// TwinCAT 3 PLC project MS
// ProgramVersion: 3.1.4024.0
// libraries:
//   Tc2_ControllerToolbox, * (Beckhoff Automation GmbH)
//   Tc2_ModbusRTU, * (Beckhoff Automation GmbH)
//   Tc2_SerialCom, * (Beckhoff Automation GmbH)
//   Tc2_Standard, * (Beckhoff Automation GmbH)
//   Tc2_System, * (Beckhoff Automation GmbH)
//   Tc2_Utilities, * (Beckhoff Automation GmbH)
//   Tc3_Module, * (Beckhoff Automation GmbH)
// project tree:
//   DATA TYPES/MODUELS/ ST_GAS_CABINET.TcDUT, ST_MAIN_MODULE.TcDUT (not stored), ST_NOTIFICATION.TcDUT (not stored), ST_NOTIFICATION_MESSAGE.TcDUT, ST_REACTOR_CABINET.TcDUT (not stored), ST_SEQUENCE.TcDUT (not stored), ST_SOL_VALVE.TcDUT, ST_TEMP_CONTROLLER.TcDUT (not stored), ST_THROTTLE_VALVE.TcDUT (not stored)
//   DATA TYPES/PARTS/ ST_ANALOG_PART.TcDUT (not stored), ST_DIGITAL_PART.TcDUT (not stored), ST_SEQUENCE_PART.TcDUT (not stored)
//   DEVICE/LINE HEATER/ FB_LINE_HEATER_MANAGER.TcPOU, FB_Modbus_Send_FIFO.TcPOU, FB_TEMP_RAMPING.TcPOU (not stored)
//   DEVICE/LINE HEATER/FUNCTION/ F_Temp_Write_Set_Point.TcPOU, F_Temp_Write_Value.TcPOU (not stored)
//   DEVICE/ ST_LineHeater_Data.TcDUT (not stored), ST_Modbus_Send_Frame.TcDUT (not stored)
//   DUTs/DUTs/ENUM/ E_aAnalogInputIO_Index.TcDUT, E_AlarmList.TcDUT (not stored), E_AlarmSetValue.TcDUT, E_InputState.TcDUT (not stored), E_Interlock.TcDUT (not stored), E_Morning_Index.TcDUT (not stored), E_WarningList.TcDUT
//   DUTs/DUTs/ F_GetReal_USINT.TcDUT (not stored)
//   DUTs/ E_ControlMode.TcDUT (not stored), E_RampGeneratorState.TcDUT (not stored), E_RecipeRun.TcDUT (not stored), E_RecipeRunETMode.TcDUT (not stored), E_TowerLamp.TcDUT (not stored), OperationMode.TcDUT, outWord.TcDUT (not stored), RampGeneratorInput.TcDUT (not stored), RecipeRunET.TcDUT (not stored), RecipeStep.TcDUT, ScaleFactor.TcDUT (not stored)
//   FUNCTION/ BOOL_TO_STRING_LHeaterON.TcPOU (not stored), CheckRangeSigned.TcPOU (not stored), CheckRangeUnsigned.TcPOU (not stored), FB_TON_Pausable.TcPOU (not stored), F_GetDorPressure.TcPOU (not stored), F_State_All_Valve_Vent.TcPOU, HEXSTR_TO_REAL_LHeaterPV.TcPOU, Real_To_String_LineHeater.TcPOU (not stored), Real_To_String_ThermalBath.TcPOU (not stored), USINT_TO_WORD_Bit.TcPOU (not stored), USINT_TO_WORD_jh.TcPOU (not stored), WORD_TO_USINT_Bit.TcPOU (not stored)
//   GVLs/ GVL_COMMAND_FROM_UI.TcGVL, GVL_CONSTANT.TcGVL (not stored), GVL_DEVICE_NET_E3508.TcGVL (not stored), GVL_DEVICE_NET_IQ_PLUS.TcGVL (not stored), GVL_IO.TcGVL (not stored), GVL.TcGVL, GVL_IO_GAS_CABINET.TcGVL (not stored), GVL_IO_REACTOR_CABINET.TcGVL (not stored), GVL_IO_VALVE.TcGVL, GVL_PERSISTENT.TcGVL, GVL_SEQUENCE.TcGVL, GVL_Serial.TcGVL, RCP.TcGVL (not stored)
//   / PlcTask.TcTTO
//   POUs/ FB_AnalogDeviceRampControl.TcPOU (not stored), FB_ControlRampGenerator.TcPOU, FB_DeviationCheck.TcPOU (not stored), FB_FaultCheck.TcPOU (not stored), FB_OverLimitCheck.TcPOU (not stored), FB_RecipeAnalogControlInputSequencer.TcPOU, F_StopAnalogRamping_ForRecipe.TcPOU (not stored), FB_SensorLimitCheck.TcPOU (not stored), FB_ValveControl.TcPOU, F_ResetTimersAndRCPTimes.TcPOU (not stored), MAIN.TcPOU, P11_E3508.TcPOU (not stored), P12_IQ_PLUS.TcPOU (not stored), P13_LineHeater.TcPOU (not stored), P14_ThermalBath.TcPOU (not stored), P15_RotationOperation.TcPOU (not stored), P16_CoverOperation.TcPOU, P17_DOROperation.TcPOU (not stored), P22_Background_ThermalBath.TcPOU (not stored), P30_ManualControl.TcPOU, P31_PriorityControl.TcPOU (not stored), P50_RecipeControl.TcPOU, P60_UpdatePV.TcPOU, P70_Interface.TcPOU, P90_Interlock.TcPOU (not stored), P91_Monitoring.TcPOU, P92_Maintenance.TcPOU (not stored)
//   POUs/FUNCTION/ FB_RINGBUFFER.TcPOU (not stored), F_StateValve_Process_Source.TcPOU (not stored), F_StateValve_Process.TcPOU (not stored)
//   POUs/VARIABLE_LINK/ F_Variable_DeviceLink.TcPOU (not stored), F_Variable_Valve.TcPOU (not stored), F_Variable_FromUI.TcPOU, F_Variable_FromUI_Interlock.TcPOU (not stored), F_Variable_TODevice.TcPOU, F_Variable_ToUI_InputState.TcPOU (not stored)

CONFIGURATION MS
    RESOURCE PLC ON TwinCAT3
        TASK PlcTask(INTERVAL := T#10ms, PRIORITY := 20);
        PROGRAM MAIN WITH PlcTask : MAIN;
    END_RESOURCE
END_CONFIGURATION

// ---- DATA TYPES/MODUELS/ST_GAS_CABINET.TcDUT
TYPE ST_GAS_CABINET :
STRUCT
	DI_01_ResetButton :ST_DIGITAL_PART;
	DI_01_GasCabinetLampButton :ST_DIGITAL_PART;
	DI_01_PneumaticPressureSensor :ST_DIGITAL_PART;
	DI_01_GasCabinetDoorClose :ST_DIGITAL_PART;
	DI_01_ControlCabinetDoorClose :ST_DIGITAL_PART;
	DI_01_SMPS_1Alarm :ST_DIGITAL_PART;
	DI_01_SMPS_2Alarm :ST_DIGITAL_PART;
	DI_01_SMPS_3Alarm :ST_DIGITAL_PART;
	
	DI_02_SMPS_4Alarm :ST_DIGITAL_PART;
	DI_02_GraphiteHeaterELCB :ST_DIGITAL_PART;
	DI_02_ThermalBathsELCB :ST_DIGITAL_PART;
	DI_02_VacuumPumpELCB :ST_DIGITAL_PART;
	DI_02_LineHeatersELCB :ST_DIGITAL_PART;
	DI_02_RotationMotorCP :ST_DIGITAL_PART;
	DI_02_CoverLiftMotorCP :ST_DIGITAL_PART;
	DI_02_T_VCP :ST_DIGITAL_PART;
	
	DI_03_GasDetectorCP :ST_DIGITAL_PART;
	DI_03_CabinetLampsCP :ST_DIGITAL_PART;
	DI_03_MFCPowerCP :ST_DIGITAL_PART;
	DI_03_LineHeater_1CP :ST_DIGITAL_PART;
	DI_03_LineHeater_2CP :ST_DIGITAL_PART;
	DI_03_LineHeater_3CP :ST_DIGITAL_PART;
	
	DI_03_LineHeater_4CP :ST_DIGITAL_PART;
	DI_03_LineHeater_5CP :ST_DIGITAL_PART;
	DI_04_LineHeater_6CP :ST_DIGITAL_PART;
	DI_04_LineHeater_7CP :ST_DIGITAL_PART;
	DI_04_LineHeater_8CP :ST_DIGITAL_PART;
	DI_04_GasDetectorH2 :ST_DIGITAL_PART;
	DI_04_GasDetectorH2S :ST_DIGITAL_PART;
	DI_04_GasDetectorH2Se :ST_DIGITAL_PART;
	DI_04_FireSensor :ST_DIGITAL_PART;
	DI_04_ExternalScrubberFault :ST_DIGITAL_PART;
	
	DI_05_ExternalH2GasCabinetFault :ST_DIGITAL_PART;
	DI_05_ExternalH2SGasCabinetFault :ST_DIGITAL_PART;
	DI_05_ExternalH2SeGasCabinetFault :ST_DIGITAL_PART;
	DI_05_ExternalUserInputAlarm :ST_DIGITAL_PART;
	DI_05_ThermalBath_1DeviationAlarm :ST_DIGITAL_PART;
	DI_05_ThermalBath_1CutOffAlarm :ST_DIGITAL_PART;
	DI_05_ThermalBath_2DeviationAlarm :ST_DIGITAL_PART;
	DI_05_ThermalBath_2CutOffAlarm :ST_DIGITAL_PART;
	
	DI_06_ThermalBath_3DeviationAlarm :ST_DIGITAL_PART;
	DI_06_ThermalBath_3CutOffAlarm :ST_DIGITAL_PART;
	DI_06_ThermalBath_4DeviationAlarm :ST_DIGITAL_PART;
	DI_06_ThermalBath_4CutOffAlarm :ST_DIGITAL_PART;
	DI_06_Spare_01 :ST_DIGITAL_PART;
	DI_06_Spare_02 :ST_DIGITAL_PART;
	DI_06_Spare_03 :ST_DIGITAL_PART;
	DI_06_Spare_04 :ST_DIGITAL_PART;
	
	DO_07_SystemPowerOffLock :ST_DIGITAL_PART;
	DO_07_GasCabinetLamp :ST_DIGITAL_PART;
	DO_07_ControlCabinetLamp :ST_DIGITAL_PART;
	DO_07_GraphiteHeaterMC :ST_DIGITAL_PART;
	DO_07_ThermalBathsMC :ST_DIGITAL_PART;
	DO_07_VacuumPumpMC :ST_DIGITAL_PART;
	DO_07_LineHeatersMC :ST_DIGITAL_PART;
	DO_07_ResetButtonLamp :ST_DIGITAL_PART;
	
	DO_08_Spare_01 :ST_DIGITAL_PART;
	DO_08_Spare_02 :ST_DIGITAL_PART;
	DO_08_Spare_03 :ST_DIGITAL_PART;
	DO_08_Spare_04 :ST_DIGITAL_PART;
	DO_08_Spare_05 :ST_DIGITAL_PART;
	DO_08_Spare_06 :ST_DIGITAL_PART;
	DO_08_Spare_07 :ST_DIGITAL_PART;
	DO_08_Spare_08 :ST_DIGITAL_PART;
	
	AI_09_M01_ChalcogenRunPV :ST_ANALOG_PART;
	AI_09_M02_MORunPV :ST_ANALOG_PART;
	AI_09_M03_H2SeSupplyPV :ST_ANALOG_PART;
	AI_09_M04_H2SSupplyPV :ST_ANALOG_PART;
	
	AO_10_M01_ChalcogenRunSV :ST_ANALOG_PART;
	AO_10_M02_MORunSV :ST_ANALOG_PART;
	AO_10_M03_H2SeSupplySV :ST_ANALOG_PART;
	AO_10_M04_H2SSupplySV :ST_ANALOG_PART;
	
	AI_11_M05_Source_1TMInSupplyPV :ST_ANALOG_PART;
	AI_11_M06_Source_2TMGaSupplyPV :ST_ANALOG_PART;
	AI_11_M07_Source_3DMSeSupplyPV :ST_ANALOG_PART;
	AI_11_M08_Source_4ChalcoSupplyPV :ST_ANALOG_PART;
	
	AO_12_M05_Source_1TMInSupplySV :ST_ANALOG_PART;
	AO_12_M06_Source_2TMGaSupplySV :ST_ANALOG_PART;
	AO_12_M07_Source_3DMSeSupplySV :ST_ANALOG_PART;
	AO_12_M08_Source_4ChalcoSupplySV :ST_ANALOG_PART;
	
	AI_13_M09_LinerPurgePV :ST_ANALOG_PART;
	AI_13_M10_HeaterPurgePV :ST_ANALOG_PART;
	AI_13_M11_ChalcogenVentPV :ST_ANALOG_PART;
	AI_13_M12_MOVentPV :ST_ANALOG_PART;
	
	AO_14_M09_LinerPurgeSV :ST_ANALOG_PART;
	AO_14_M10_HeaterPurgeSV :ST_ANALOG_PART;
	AO_14_M11_ChalcogenVentSV :ST_ANALOG_PART;
	AO_14_M12_MOVentSV :ST_ANALOG_PART;
	
	AI_15_E01Source_1TMInPressurePV :ST_ANALOG_PART;
	AI_15_E02Source_2TMGaPressurePV :ST_ANALOG_PART;
	AI_15_E03Source_3DMSePressurePV :ST_ANALOG_PART;
	AI_15_E04Source_4ChalcoPressurePV :ST_ANALOG_PART;
	
	AO_16_E01Source_1TMInPressureSV :ST_ANALOG_PART;
	AO_16_E02Source_2TMGaPressureSV :ST_ANALOG_PART;
	AO_16_E03Source_3DMSePressureSV :ST_ANALOG_PART;
	AO_16_E04Source_4ChalcoPressureSV :ST_ANALOG_PART;
	
	DI_17_DP1ChalcogenDP :ST_ANALOG_PART;
	DI_17_DP2MODP :ST_ANALOG_PART;
	
	DI_18_S01N2SupplyPressPV :ST_ANALOG_PART;
	DI_18_S02H2SupplyPressPV :ST_ANALOG_PART;
	DI_18_S03H2SSupplyPressPV :ST_ANALOG_PART;
	DI_18_S04H2SeSupplyPressPV :ST_ANALOG_PART;
	
	DI_19_LineHeaterController :ST_DIGITAL_PART;
	DI_20_ThermalBathx4EA :ST_DIGITAL_PART;

END_STRUCT
END_TYPE

// ---- DATA TYPES/MODUELS/ST_NOTIFICATION_MESSAGE.TcDUT
TYPE ST_NOTIFICATION_MESSAGE :
STRUCT
	INDEX:DINT;
	TITLE:STRING(255);
	MESSAGE :STRING(255);
	NOTIFICATION_TYPE:DINT; (* NOTIFI_INTERLOCK = 1, NOTIFI_ALARM = 2, NOTIFI_MESSAGE = 3 *)
	MODULE_ID:DINT;
END_STRUCT
END_TYPE

// ---- DATA TYPES/MODUELS/ST_SOL_VALVE.TcDUT
TYPE ST_SOL_VALVE :
STRUCT
	DO_00_V01ChalcogenCarrierChange :ST_DIGITAL_PART;
	DO_00_V02MOCarreirChange :ST_DIGITAL_PART;
	DO_00_V03H2SeSourceChange :ST_DIGITAL_PART;
	DO_00_V04H2SSourceChange :ST_DIGITAL_PART;
	DO_00_V05Source_1TMInCarrierChange :ST_DIGITAL_PART;
	DO_00_V06Source_1TMInBypass :ST_DIGITAL_PART;
	DO_00_V07Source_2TMGaCarrierChange :ST_DIGITAL_PART;
	DO_00_V08Source_2TMGaBypass :ST_DIGITAL_PART;
	
	DO_00_V09Source_3DMSeCarrierChange :ST_DIGITAL_PART;
	DO_00_V10Source_3DMSeBypass :ST_DIGITAL_PART;
	DO_00_V11Source_4ChalcogenCarrierChange :ST_DIGITAL_PART;
	DO_00_V12Source_4ChalcogenBypass :ST_DIGITAL_PART;
	DO_00_V13ReactorPurgeCarrierChange :ST_DIGITAL_PART;
	DO_00_V14Source_1TMInManifoldRun :ST_DIGITAL_PART;
	DO_00_V15Source_2TMGaManifoldRun :ST_DIGITAL_PART;
	DO_00_V16Source_3DMSeManifoldRun :ST_DIGITAL_PART;
	
	DO_00_V17GasH2SeManifoldRun :ST_DIGITAL_PART;
	DO_00_V18GasH2SManifoldRun :ST_DIGITAL_PART;
	DO_00_V19Source_4ChalcogenManifoldRun :ST_DIGITAL_PART;
	DO_00_V20VentPress_Change :ST_DIGITAL_PART;
	DO_00_V21PumpByPass :ST_DIGITAL_PART;
	DO_00_V22DORVaccumON :ST_DIGITAL_PART;
	DO_00_V23DORFilling :ST_DIGITAL_PART;
	DO_00_V24Source_1LeakTest_IN :ST_DIGITAL_PART;
	
	DO_00_V25Source_1LeakTest_OUT :ST_DIGITAL_PART;
	DO_00_V26Source_2LeakTest_IN :ST_DIGITAL_PART;
	DO_00_V27Source_2LeakTest_OUT :ST_DIGITAL_PART;
	DO_00_V28Source_3LeakTest_IN :ST_DIGITAL_PART;
	DO_00_V29Source_3LeakTest_OUT :ST_DIGITAL_PART;
	DO_00_V30Source_4LeakTest_IN :ST_DIGITAL_PART;
	DO_00_V31Source_4LeakTest_OUT :ST_DIGITAL_PART;
	DO_00_V32SourceVacuumON :ST_DIGITAL_PART;
	
END_STRUCT
END_TYPE

// ---- DUTs/DUTs/ENUM/E_aAnalogInputIO_Index.TcDUT
{attribute 'qualified_only'}
{attribute 'strict'}
{attribute 'to_string'}
TYPE E_aAnalogInputIO_Index :
(
	E_PV_MFC_01 :=1,
	E_PV_MFC_02 :=2,
	E_PV_MFC_03 :=3,
	E_PV_MFC_04 :=4,
	E_PV_MFC_05 :=5,
	E_PV_MFC_06 :=6,
	E_PV_MFC_07 :=7,
	E_PV_MFC_08 :=8,
	E_PV_MFC_09 :=9,
	E_PV_MFC_10 :=10,
	E_PV_MFC_11 :=11,
	E_PV_MFC_12 :=12,
	E_PV_EPC_01 :=13,
	E_PV_EPC_02 :=14,
	E_PV_EPC_03 :=15,
	E_PV_EPC_04 :=16,
	E_PV_Susceptor_Temp:=17,
	E_PV_Reactor_Pressure:=18,
	E_PV_susceptorRotation:=19,
	E_PV_Ultimate_Pressure:=20,
	E_PV_Exhaust_Pressure:=21,
	E_PV_DOR_PRESSURE:=22,
	E_PV_GAS_Pressure_N2:=23,
	E_PV_GAS_Pressure_H2:=24,
	E_PV_GAS_Pressure_H2S:=25,
	E_PV_GAS_Pressure_H2Se:=26,
	E_PV_CoolingWafer_SH:=27
);
END_TYPE

// ---- DUTs/DUTs/ENUM/E_AlarmSetValue.TcDUT
{attribute 'qualified_only'}
{attribute 'strict'}
{attribute 'to_string'}
TYPE E_AlarmSetValue :
(
//	E_AS_Alarm_Deviation:=1,
//	E_AS_Warning_Deviation,
//	E_AS_DelayTime_Analog,
//	E_AS_DelayTime_Digital,
//	E_AS_Process_Gas_Pressure_Alarm,
//	E_AS_Process_Gas_Pressure_Warning,
//	E_AS_CWTemp_SH_ALARM,
//	E_AS_CWTemp_SH_WARNING,
//	E_AS_CWTemp_COIL_ALARM,
//	E_AS_CWTemp_COIL_WARNING,
//	E_AS_SUSCEPTOR_OVER_TEMP,
//	E_AS_REACTOR_OVRE_PRESSURE,
//	E_AS_CAN_OPEN_TEMP,
//	E_AS_CAN_OPEN_REACTOR_PRESSURE,
//	E_AS_DOR_Pressure_Limit,
//	E_AS_DOR_RerayCount,
	E_AS_END
);
END_TYPE

// ---- DUTs/DUTs/ENUM/E_WarningList.TcDUT
{attribute 'qualified_only'}
{attribute 'strict'}
{attribute 'to_string'}
TYPE E_WarningList :
(
	E_WarningList_GasPressure_Low_N2:=1,
	E_WarningList_GasPressureLowN2,
	E_WarningList_GasPressureLowH2,
	E_WarningList_GasPressureLowNH3,
	E_WarningList_GasPressureLowSiH4,
	E_WarningList_CWTemperatureHighSH,
	E_WarningList_CWTemperatureHighCoil,
	E_WarningList_SusceptorOverTemperature,
	E_WarningList_ReactorOverPressure,
	E_WarningList_PneumaticPressureLow,
	E_WarningList_CoolingWaterLow,
	E_WarningList_InductionHeaterFault,
	E_WarningList_RotationMotorFault,
	E_WarningList_VacuumPumpFault,
	E_WarningList_GasCabinetDoorOpen,
	E_WarningList_ReactorCabinetDoorOpen,
	E_WarningList_SusceptorTemperatureDeviation,
	E_WarningList_ReactorPressureDeviation,
	E_WarningList_SusceptorRotationDeviation,
	E_WarningList_MORunDeviation,
	E_WarningList_HydRunDeviation,
	E_WarningList_NH3LargeINDeviation,
	E_WarningList_NH3SmallINDeviation,
	E_WarningList_SiHINDeviation,
	E_WarningList_SiHDilutionDeviation,
	E_WarningList_SiHDilutedDeviation,
	E_WarningList_TEBBubblingDeviation,
	E_WarningList_TMAlBubblingDeviation,
	E_WarningList_TMInBubblingDeviation,
	E_WarningList_TMGaBubblingDeviation,
	E_WarningList_DTMGaBubblingDeviation,
	E_WarningList_DTMGaDilutionDeviation,
	E_WarningList_DTMGaDilutedDeviation,
	E_WarningList_Cp2MgBubblingDeviation,
	E_WarningList_ReactorPurgeDeviation,
	E_WarningList_RotationSealPurgeDeviation,
	E_WarningList_MOVentDeviation,
	E_WarningList_HydVentDeviation,
	E_WarningList_SiH4PressureDeviation,
	E_WarningList_TEBPressureDeviation,
	E_WarningList_TMAlPressureDeviation,
	E_WarningList_TMInPressureDeviation,
	E_WarningList_TMGaPressureDeviation,
	E_WarningList_DTMGaPressureDeviation,
	E_WarningList_Cp2MgPressureDeviation,
	E_WarningList_END

);
END_TYPE

// ---- DUTs/OperationMode.TcDUT
{attribute 'qualified_only'}
{attribute 'strict'}
{attribute 'to_string'}
TYPE OperationMode :
(
	Manual := 0,
	Recipe := 1,
	Priority := 2
);
END_TYPE

// ---- DUTs/RecipeStep.TcDUT
TYPE RecipeStep :
STRUCT
	sRecipe : STRING(81);
	iRecipe : ARRAY[1..5] OF INT; //Reactor Condition
	rRecipe : ARRAY[1..GVL_CONSTANT.NumAnalogController] OF REAL; //MFC, EPC Data
	cTemp 	: REAL := 0; 	
	dRecipe : DWORD; //Valve Data
END_STRUCT
END_TYPE

// ---- GVLs/GVL_COMMAND_FROM_UI.TcGVL
{attribute 'qualified_only'}
VAR_GLOBAL
	
	//GVL_IO.aOutputCmd[1].
	
	CMD_HEATER_MAIN_MC_ON:BOOL;  //[1].0
	CMD_THERMAL_BACH_MC_ON:BOOL;//[1].1
	CMD_VACUUM_PUMP_MC_ON:BOOL;//[1].2
	CMD_LINE_HEATER_MC_ON:BOOL;//[1].3
	CMD_SPARE_1_4:BOOL;//[1].4
	CMD_SPARE_1_5:BOOL;//[1].5
	CMD_VACUUM_PUMP_ON:BOOL;//[1].6
	CMD_VACUUM_PUMP_RESET:BOOL;//[1].7
	CMD_ROTATION_START:BOOL;//[1].8
	CMD_ROTATION_RESET:BOOL;//[1].9
	CMD_MAIN_POWER_RESET:BOOL;//[1].10
	
	CMD_E3508_MAN_AUTO:BOOL;//[1].11
	CMD_THROTTLE_PRESSURE_POSITION_MODE:BOOL;//[1].12
	CMD_THROTTLE_OUTPUT_MODE:USINT;//[2]	
END_VAR

// ---- GVLs/GVL.TcGVL
{attribute 'qualified_only'}
VAR_GLOBAL
	MainModule:ST_MAIN_MODULE;
	fbLineHeater_Manager:FB_LINE_HEATER_MANAGER;
	
	RotationResetTon: TON;
END_VAR

// ---- GVLs/GVL_IO_VALVE.TcGVL
{attribute 'qualified_only'}
VAR_GLOBAL
	DO_00_V01ChalcogenCarrierChange AT%Q*:BOOL;
	DO_00_V02MOCarreirChange AT%Q*:BOOL;
	DO_00_V03H2SeSourceChange AT%Q*:BOOL;
	DO_00_V04H2SSourceChange AT%Q*:BOOL;
	DO_00_V05Source_1TMInCarrierChange AT%Q*:BOOL;
	DO_00_V06Source_1TMInBypass AT%Q*:BOOL;
	DO_00_V07Source_2TMGaCarrierChange AT%Q*:BOOL;
	DO_00_V08Source_2TMGaBypass AT%Q*:BOOL;
	DO_00_V09Source_3DMSeCarrierChange AT%Q*:BOOL;
	DO_00_V10Source_3DMSeBypass AT%Q*:BOOL;
	DO_00_V11Source_4ChalcogenCarrierChange AT%Q*:BOOL;
	DO_00_V12Source_4ChalcogenBypass AT%Q*:BOOL;
	DO_00_V13ReactorPurgeCarrierChange AT%Q*:BOOL;
	DO_00_V14Source_1TMInManifoldRun AT%Q*:BOOL;
	DO_00_V15Source_2TMGaManifoldRun AT%Q*:BOOL;
	DO_00_V16Source_3DMSeManifoldRun AT%Q*:BOOL;
	DO_00_V17GasH2SeManifoldRun AT%Q*:BOOL;
	DO_00_V18GasH2SManifoldRun AT%Q*:BOOL;
	DO_00_V19Source_4ChalcogenManifoldRun AT%Q*:BOOL;
	DO_00_V20VentPress_Change AT%Q*:BOOL;
	DO_00_V21PumpByPass AT%Q*:BOOL;
	DO_00_V22DORVaccumON AT%Q*:BOOL;
	DO_00_V23DORFilling AT%Q*:BOOL;
	DO_00_V24Source_1LeakTest_IN AT%Q*:BOOL;
	DO_00_V25Source_1LeakTest_OUT AT%Q*:BOOL;
	DO_00_V26Source_2LeakTest_IN AT%Q*:BOOL;
	DO_00_V27Source_2LeakTest_OUT AT%Q*:BOOL;
	DO_00_V28Source_3LeakTest_IN AT%Q*:BOOL;
	DO_00_V29Source_3LeakTest_OUT AT%Q*:BOOL;
	DO_00_V30Source_4LeakTest_IN AT%Q*:BOOL;
	DO_00_V31Source_4LeakTest_OUT AT%Q*:BOOL;
	DO_00_V32SourceVacuumON AT%Q*:BOOL;
END_VAR

// ---- GVLs/GVL_PERSISTENT.TcGVL
{attribute 'qualified_only'}
VAR_GLOBAL PERSISTENT
	parameter_Test:INT;
	parameter_Test_1:INT;
	parameter_Test_2:INT;
END_VAR

// ---- GVLs/GVL_SEQUENCE.TcGVL
{attribute 'qualified_only'}
VAR_GLOBAL
//	fbUpdateModue:FB_UPDATE_MODULE;
	
	fbDeviationCheck		:ARRAY[1..29] OF FB_DeviationCheck;
	fbDeviationCheck_Reactor		:ARRAY[1..3] OF FB_DeviationCheck;
	fbSensorLimitCheck		:ARRAY[1..4] OF FB_SensorLimitCheck;  // Pressure N2 H2 H2S,H2SE 
	fbSensorOverLimitCheck	:ARRAY[1..2] OF FB_OverLimitCheck;  // Over Temp  , Over Pressure  
	fbFaultCheck			:ARRAY[1..8] OF FB_FaultCheck; // CDA/CoolingWafer/Rotation Fault/Vacuum Pump Fault/Gas Cabinet Open / Reactor Door Open / Dor Fault
	fbFaultCheck_Utility	:ARRAY[1..4] OF FB_FaultCheck; //SMPS,Circuit Power , Gas Detector , External Alarm
	fbFaultCheck_Utility_CP :ARRAY[1..4] OF FB_FaultCheck; //CP
	
	FB_DOR_PRESSURE_AVG: FB_RINGBUFFER;
	FB_EXHAUST_AVG: FB_RINGBUFFER;
END_VAR

// ---- GVLs/GVL_Serial.TcGVL
{attribute 'qualified_only'}
VAR_GLOBAL
	TxBufferTB : ComBuffer; (* Receive data buffer; used with all receive function blocks *)
	RxBufferTB : ComBuffer; (* Transmit data buffer; used with all receive function blocks *)
	
	stIn_KL6031_TB AT %I*	: KL6inData22B;	(* linked to the KL6001 in the TwinCAT System Manager *)
	stOut_KL6031_TB AT %Q*	: KL6outData22B;	(* linked to the KL6001 in the TwinCAT System Manager *)	
	
	LineHeater_data_1	:ST_LineHeater_Data;
	LineHeater_data_2	:ST_LineHeater_Data;
END_VAR

// ---- POUs/MAIN.TcPOU
PROGRAM MAIN
VAR_INPUT
	controlModeCmd : E_ControlMode := E_ControlMode.Manual;
END_VAR
VAR
	controlMode	: E_ControlMode := controlModeCmd;
	prevControlMode : E_ControlMode := controlMode;
END_VAR

F_Variable_Valve();
F_Variable_DeviceLink();
F_Variable_FromUI();
F_Variable_FromUI_Interlock();
F_Variable_TODevice();
F_Variable_ToUI_InputState();
GVL.fbLineHeater_Manager(RData_Module_1=>GVL_Serial.LineHeater_data_1,RData_Module_2=>GVL_Serial.LineHeater_data_2);


P11_E3508(); //Temp Controller
P12_IQ_PLUS(); //Throttle Valve Controller
P13_LineHeater();
P14_ThermalBath();
P15_RotationOperation();
P16_CoverOperation();
P17_DOROperation();
P22_Background_ThermalBath();


IF controlMode <> E_ControlMode.Priority THEN
	IF controlMode <> controlModeCmd THEN
		IF controlModeCmd = E_ControlMode.Priority THEN
			prevControlMode := controlMode;
		END_IF
		controlMode := controlModeCmd;
	END_IF
END_IF

CASE controlMode OF
	E_ControlMode.Manual:
		P30_ManualControl();
	
	E_ControlMode.Recipe:
		P50_RecipeControl(); //레시피 콘트론
		
	E_ControlMode.Priority:
		P31_PriorityControl();
		IF P31_PriorityControl.complete = TRUE THEN
			controlMode := prevControlMode;
			controlModeCmd := controlMode;
		END_IF
END_CASE

P60_UpdatePV();
P70_Interface();
P90_Interlock();
P91_Monitoring();
P92_Maintenance();

END_PROGRAM

// ---- POUs/VARIABLE_LINK/F_Variable_FromUI.TcPOU
FUNCTION F_Variable_FromUI: BOOL


VAR
	rRotationAlarm_Reset: R_TRIG;
	
	Rotation_Shift: WORD;
END_VAR

////UI에서 Write하는 Command
//아래 MC는 Maint 모드에서만 조작 가능
//GVL_COMMAND_FROM_UI.CMD_HEATER_MAIN_MC_ON:= GVL_IO.aOutputCmd[1].0;
//GVL_COMMAND_FROM_UI.CMD_THERMAL_BACH_MC_ON:= GVL_IO.aOutputCmd[1].1;
//GVL_COMMAND_FROM_UI.CMD_VACUUM_PUMP_MC_ON:= GVL_IO.aOutputCmd[1].2;
//GVL_COMMAND_FROM_UI.CMD_LINE_HEATER_MC_ON := GVL_IO.aOutputCmd[1].3;

GVL_COMMAND_FROM_UI.CMD_VACUUM_PUMP_ON := GVL_IO.aOutputCmd[1].6;
GVL_COMMAND_FROM_UI.CMD_VACUUM_PUMP_RESET:= GVL_IO.aOutputCmd[1].7;

GVL_COMMAND_FROM_UI.CMD_ROTATION_START:= GVL_IO.aOutputCmd[1].8;
GVL_COMMAND_FROM_UI.CMD_ROTATION_RESET := GVL_IO.aOutputCmd[1].10;

//jhkang 하드웨어로 구성 되어 있어야 하는데 아직 구성 안됨 := GVL_IO.aOutputCmd[1].10;
GVL_COMMAND_FROM_UI.CMD_E3508_MAN_AUTO := GVL_IO.aOutputCmd[1].12;(*True:Manual  False:auto*)
GVL_COMMAND_FROM_UI.CMD_THROTTLE_PRESSURE_POSITION_MODE := GVL_IO.aOutputCmd[1].13;//true: Pressure False:Position

GVL_COMMAND_FROM_UI.CMD_THROTTLE_OUTPUT_MODE:= WORD_TO_USINT(GVL_IO.aOutputCmd[2]); //Throttle Valve Mode Setting 0:Normal 1:Close 2:Open 3:Hold 4:Reset

GVL_IO_GAS_CABINET.DO_07_GraphiteHeaterMC :=  GVL_COMMAND_FROM_UI.CMD_HEATER_MAIN_MC_ON;
GVL_IO_GAS_CABINET.DO_07_ThermalBathsMC :=  GVL_COMMAND_FROM_UI.CMD_THERMAL_BACH_MC_ON;
GVL_IO_GAS_CABINET.DO_07_VacuumPumpMC :=  GVL_COMMAND_FROM_UI.CMD_VACUUM_PUMP_MC_ON;
GVL_IO_GAS_CABINET.DO_07_LineHeatersMC:=  GVL_COMMAND_FROM_UI.CMD_LINE_HEATER_MC_ON;

//GVL_IO_REACTOR_CABINET.DO_05_SusceptorRotationFWD:=GVL_COMMAND_FROM_UI.CMD_ROTATION_START;

rRotationAlarm_Reset(CLK:=GVL_COMMAND_FROM_UI.CMD_ROTATION_RESET);
IF rRotationAlarm_Reset.Q THEN
	GVL_IO_REACTOR_CABINET.DO_05_SusceptorRotationAL_RST:=TRUE;
END_IF

GVL.RotationResetTon(IN:=GVL_IO_REACTOR_CABINET.DO_05_SusceptorRotationAL_RST,PT:=T#3S);

IF GVL_IO_REACTOR_CABINET.DI_02_SusceptorRotationMotorFault = TRUE OR GVL.RotationResetTon.Q THEN
	GVL.RotationResetTon(in:=FALSE);
	IF GVL_IO_REACTOR_CABINET.DO_05_SusceptorRotationAL_RST = TRUE THEN
		GVL_IO_REACTOR_CABINET.DO_05_SusceptorRotationAL_RST:=FALSE;
	END_IF
	
	IF GVL_IO.aOutputCmd[1].10 = TRUE THEN
		GVL_IO.aOutputCmd[1].10:=FALSE;
	END_IF
END_IF


	//GVL_IO_REACTOR_CABINET.DO_05_SusceptorRotationAL_RST:=GVL_COMMAND_FROM_UI.CMD_ROTATION_RESET;	
GVL_IO_REACTOR_CABINET.DO_05_VacuumPumpStart_Stop := GVL_COMMAND_FROM_UI.CMD_VACUUM_PUMP_ON;
GVL_IO_REACTOR_CABINET.DO_05_VacuumPumpReset:=GVL_COMMAND_FROM_UI.CMD_VACUUM_PUMP_RESET;

END_FUNCTION

// ---- POUs/VARIABLE_LINK/F_Variable_TODevice.TcPOU
FUNCTION F_Variable_TODevice: BOOL

;

END_FUNCTION

// ---- POUs/P16_CoverOperation.TcPOU
PROGRAM P16_CoverOperation
VAR
// 	isCoverClosed 	: BOOL;

	bCoverCP	: BOOL;
	bLowerLimit	: BOOL;
	bUpperLimit	: BOOL;
	TimerUpLED 		: TON;
	TimerUpLED_X 	: TON;
	TimerDownLED 	: TON;
	TimerDownLED_X 	: TON;
	TimerDownDelayOff 	: TON;
	(* Input *)
	bUpSwitch	: BOOL;
	bDownSwitch 	: BOOL;
	bClamp_Lock_switch: BOOL;
	bClamp_Release_switch: BOOL;
	(* Output *)
	bUpLED 		: BOOL;
	bDownLED 	: BOOL;
	bOnUpRelay 	: BOOL;
	bOnDownRelay : BOOL;
	bOnClamp_Lock_Relay:BOOL;
	bOnClamp_Release_Relay:BOOL;		
	
	bClampLock: BOOL;
	bClampRelease: BOOL;
END_VAR

_DigitalInput();

TimerDownDelayOff(IN:=bLowerLimit, PT:=T#500MS);

//Cover Open 조건
//공정 중이지 않을것
//Dor Pressure down
//Clamp Releaae
//Susceptor down
//CDG 700 torr 이상
//모든 벨브 ff

// Cover Operation Condition
IF P90_Interlock.bReactorOpenEnable THEN
	(*Cover*)
	IF bClampRelease THEN
		bOnUpRelay := (bDownSwitch = FALSE AND bUpSwitch = TRUE AND bUpperLimit = FALSE );
		bOnDownRelay := (bDownSwitch = TRUE AND bUpSwitch = FALSE AND (bLowerLimit = FALSE OR TimerDownDelayOff.Q = FALSE ));
	ELSE
		bOnUpRelay:=FALSE;
		bOnDownRelay:=FALSE;
	END_IF
	(*clamp*)
	bOnClamp_Lock_Relay:=(bClamp_Lock_switch = TRUE AND bClamp_Release_switch = FALSE);
	bOnClamp_Release_Relay:=(bClamp_Lock_switch = FALSE AND bClamp_Release_switch = TRUE);
ELSE
	(*Cover*)
	bOnUpRelay:=FALSE;
	bOnDownRelay:=FALSE;
	(*clamp*)
	bOnClamp_Lock_Relay:=FALSE;
	bOnClamp_Release_Relay:=FALSE;
END_IF

//LED Blinking
TimerUpLED(IN:=(bOnUpRelay AND TimerUpLED_X.Q = FALSE), PT:=T#500MS);
TimerUpLED_X(IN:=TimerUpLED.Q, PT:=T#300MS);
bUpLED := (TimerUpLED.Q AND bOnUpRelay) OR bUpperLimit;

TimerDownLED(IN:=(bOnDownRelay AND TimerDownLED_X.Q = FALSE), PT:=T#500MS);
TimerDownLED_X(IN:=TimerDownLED.Q, PT:=T#300MS);
bDownLED := (TimerDownLED.Q AND bOnDownRelay) OR bLowerLimit;

_DigitalOutput();

ACTION _DigitalInput:
//(* Read from Device Value *)
//// Cover Operation Switch

bUpSwitch 		:=GVL_IO_REACTOR_CABINET.DI_01_ReactorDoorUpButton;
bDownSwitch 	:=GVL_IO_REACTOR_CABINET.DI_01_ReactorDoorDownButton;
bUpperLimit 	:=GVL_IO_REACTOR_CABINET.DI_02_ReactorDoorUpLimitSensor;
bLowerLimit 	:=GVL_IO_REACTOR_CABINET.DI_03_ReactorDoorDownLimitSensor;
bCoverCP 		:= GVL_IO_GAS_CABINET.DI_02_CoverLiftMotorCP;

bClampLock := GVL_IO_REACTOR_CABINET.DI_03_CylinderAutoSwitch_Closed;
bClampRelease :=GVL_IO_REACTOR_CABINET.DI_03_CylinderAutoSwitch_Opened;

bClamp_Lock_switch:=GVL_IO_REACTOR_CABINET.DI_01_ClampLock;
bClamp_Release_switch:=GVL_IO_REACTOR_CABINET.DI_01_ClampRelease;
END_ACTION

ACTION _DigitalOutput:
(* Write to Device Value *)
// Cover Operation Switch Lamp


//Status Output
GVL_IO.isCoverClosed := bLowerLimit;

GVL_IO_REACTOR_CABINET.DO_06_ReactorCoverUpButtonLamp := bUpLED;
GVL_IO_REACTOR_CABINET.DO_06_ReactorCoverDownButtonLamp := bDownLED;

GVL_IO_REACTOR_CABINET.DO_04_ReactorCoverUpRelay :=bOnUpRelay;
GVL_IO_REACTOR_CABINET.DO_04_ReactorCoverDownRelay :=bOnDownRelay;

GVL_IO_REACTOR_CABINET.DO_06_ClampLockButtonLamp := GVL_IO_REACTOR_CABINET.DI_03_CylinderAutoSwitch_Closed;
GVL_IO_REACTOR_CABINET.DO_06_ClampReleaseButtonLamp := GVL_IO_REACTOR_CABINET.DI_03_CylinderAutoSwitch_Opened;

GVL_IO_REACTOR_CABINET.DO_05_ClampLock := bOnClamp_Lock_Relay;
GVL_IO_REACTOR_CABINET.DO_05_ClampRelease := bOnClamp_Release_Relay;
END_ACTION

END_PROGRAM

// ---- POUs/P30_ManualControl.TcPOU
Program P30_ManualControl
VAR
	analogDeviceRampControl : FB_AnalogDeviceRampControl;
END_VAR

analogDeviceRampControl();

END_PROGRAM

// ---- POUs/P50_RecipeControl.TcPOU
PROGRAM P50_RecipeControl
VAR
	nRcpIndex		: INT;
	eRecipeRun		: E_RecipeRun ; //레시피 상태
	fbAnalogDeviceRampControl : FB_AnalogDeviceRampControl;
	fbRecipeAnalogInputControlSequencer: FB_RecipeAnalogControlInputSequencer;
	fbValveControl: FB_ValveControl;
	
	Pause_TON		: TON;
	Ramp_TON		: FB_TON_Pausable;
	Hold_TON		: FB_TON_Pausable;
	
	loopCount		: ARRAY[1..100] OF INT;
	i				: INT;
END_VAR
VAR CONSTANT
	Pause_MAX		: TIME := T#1800S;
END_VAR

CASE RCP.cmd_RcpOperation OF
	0: //Init State
 		f_ResetTimersAndRCPTimes(fbPause_TON := Pause_TON, fbRamp_TON := Ramp_TON, fbHold_TON := Hold_TON);
		
		FOR i:=1 TO Rcp.iRcpTotalStep DO
			loopCount[i] := Rcp.aRecipe[i].iRecipe[5];
		END_FOR
		
		nRcpIndex := 0;
		Rcp.userState := 0;
		eRecipeRun := E_RecipeRun.Initial;
		GVL_IO.nCaseSignalTower := 5; // White - Idle

	10: //RUN
		IF nRcpIndex = 0 THEN
			nRcpIndex := 1;
		END_IF
		fbAnalogDeviceRampControl();
						
		// CASE 문을 이용한 상태 머신 구현
		CASE eRecipeRun OF
			E_RecipeRun.Initial:
				f_ResetTimersAndRCPTimes(fbPause_TON := Pause_TON, fbRamp_TON := Ramp_TON, fbHold_TON := Hold_TON);
				fbRecipeAnalogInputControlSequencer(rRecipe := RCP.aRecipe[nRcpIndex].rRecipe, rampTime:= TO_UINT(RCP.aRecipe[nRcpIndex].iRecipe[2]));
				fbValveControl(valveSetting:= RCP.aRecipe[nRcpIndex].dRecipe);
				Rcp.userState := 10;// Recipe Running
				GVL_IO.nCaseSignalTower := 3;
				eRecipeRun := E_RecipeRun.Ramp;
				
			E_RecipeRun.Ramp: // Ramp 수행
				Ramp_TON(IN:=TRUE, PT:= RCP.aRecipe[nRcpIndex].iRecipe[2] * T#1S, ET=>RCP.RecipeRunET.ET);
				RCP.RecipeRunET.Mode := E_RecipeRunETMode.Ramp;
				IF Ramp_TON.Q THEN
					Ramp_TON(IN:=FALSE);
					eRecipeRun := E_RecipeRun.CheckHoldTemp;
				END_IF				
				
			E_RecipeRun.CheckHoldTemp: //Hold Temp 확인
				IF RCP.aRecipe[nRcpIndex].cTemp = 0.0 THEN
					Hold_TON(IN:=TRUE, PT:= RCP.aRecipe[nRcpIndex].iRecipe[3] * T#1S, ET=>RCP.RecipeRunET.ET);
					RCP.RecipeRunET.Mode := E_RecipeRunETMode.Hold;
					IF Hold_TON.Q THEN
						Hold_TON(IN:=FALSE);
						eRecipeRun := E_RecipeRun.End; // 레시피 첫 Column 실행
					END_IF
				ELSIF GVL_IO.aController_PV[E_aAnalogInputIO_Index.E_PV_Susceptor_Temp] < RCP.aRecipe[nRcpIndex].cTemp THEN //서셉터 온도가 Wait 온도보다 낮을 때
					Hold_TON(IN:=FALSE);
					eRecipeRun := E_RecipeRun.End; // 레시피 첫 Column 실행
				ELSE // 서셉터 온도가 Wait 온도보다 높을 때
					;// 떨어질 때까지 기다림
				END_IF
				
			E_RecipeRun.End: // 다음 Step 이동 (루프 마지막 단계일 경우, 다음 Step 이동 또는 루프 처음단계로 점프)
				loopCount[nRcpIndex] := loopCount[nRcpIndex] - 1;
				nRcpIndex := nRcpIndex + 1 - (RCP.aRecipe[nRcpIndex].iRecipe[4]) * MIN(loopCount[nRcpIndex], 1);
				IF nRcpIndex > Rcp.iRcpTotalStep THEN
					RCP.cmd_RcpOperation := 50;
				END_IF
				eRecipeRun := E_RecipeRun.Initial;
		END_CASE
		
	20: //PAUSE
		CASE eRecipeRun OF
			E_RecipeRun.Ramp:
				Ramp_TON(PAUSE:=TRUE);		
			E_RecipeRun.CheckHoldTemp:
				Hold_TON(PAUSE:=TRUE);
		END_CASE
		
		Pause_TON(IN:=TRUE, PT:= Pause_MAX, ET=>RCP.Pause_ET); //최대 홀드 시간이 지나면 다음 스텝으로 넘거감
		IF Pause_TON.Q THEN
			Pause_TON(IN:=FALSE);
			eRecipeRun := E_RecipeRun.End; // 레시피 첫 Column 실행
		END_IF

		Rcp.userState := 20;
		GVL_IO.nCaseSignalTower := 5;
		
	30: //RESTART
		Pause_TON(IN:=FALSE);
		CASE eRecipeRun OF
			E_RecipeRun.Ramp:
				Ramp_TON(PAUSE:=FALSE);
			
			E_RecipeRun.CheckHoldTemp:
				Hold_TON(PAUSE:=FALSE);
		END_CASE

		RCP.Pause_ET := T#0S;
		Rcp.userState := 10;
		RCP.cmd_RcpOperation := 10;	
		GVL_IO.nCaseSignalTower := 3;
		
	40: //STOP
		f_ResetTimersAndRCPTimes(fbPause_TON := Pause_TON, fbRamp_TON := Ramp_TON, fbHold_TON := Hold_TON);
		F_StopAnalogRamping_ForRecipe();
		Rcp.userState := 40;
		GVL_IO.nCaseSignalTower := 5;
		
	50: //END
		f_ResetTimersAndRCPTimes(fbPause_TON := Pause_TON, fbRamp_TON := Ramp_TON, fbHold_TON := Hold_TON);
		Rcp.userState := 50;
		fbAnalogDeviceRampControl();
		GVL_IO.nCaseSignalTower := 5;
		
	60: //SKIP
		IF E_RecipeRun.Ramp <= eRecipeRun  AND  eRecipeRun <= E_RecipeRun.CheckHoldTemp THEN
			eRecipeRun := E_RecipeRun.End;
		END_IF
		Rcp.cmd_RcpOperation := 10;
		RCP.Pause_ET := T#0S;
END_CASE
RCP.iRcpStepN := nRcpIndex;

END_PROGRAM

// ---- POUs/FB_RecipeAnalogControlInputSequencer.TcPOU
FUNCTION_BLOCK FB_RecipeAnalogControlInputSequencer
VAR_INPUT
	rampTime: UINT;
END_VAR
VAR_IN_OUT
	rRecipe: ARRAY[1..(GVL_CONSTANT.NumAnalogController)] OF REAL;
END_VAR
VAR
	i: INT;
END_VAR

FOR i:= 1 TO E_aAnalogInputIO_Index.E_PV_EPC_04 DO
	IF 0.0 < GVL_IO.aMaxValueController[i] THEN
		GVL_IO.aController[i].input.restart := TRUE;
		GVL_IO.aController[i].input.rampTime := rampTime; 
		GVL_IO.aController[i].input.targetValue := rRecipe[i] / GVL_IO.aMaxValueController[i] * GVL_CONSTANT.EL3064MaxValueH;
	END_IF
END_FOR

FOR i:= E_aAnalogInputIO_Index.E_PV_Susceptor_Temp TO E_aAnalogInputIO_Index.E_PV_susceptorRotation DO
	GVL_IO.aController[i].input.restart := TRUE;
	GVL_IO.aController[i].input.rampTime := rampTime;
	GVL_IO.aController[i].input.targetValue := rRecipe[i];
END_FOR

END_FUNCTION_BLOCK

// ---- POUs/FB_ValveControl.TcPOU
FUNCTION_BLOCK FB_ValveControl
VAR_INPUT
	valveSetting: DWORD; 
END_VAR

(* Solenoid Valve Mapping *)
GVL_IO.aOutputSolValve.0 := valveSetting.0; //V01 B/G N2 In
GVL_IO.aOutputSolValve.1 := valveSetting.1;
GVL_IO.aOutputSolValve.2 := valveSetting.2;
GVL_IO.aOutputSolValve.3 := valveSetting.3;
GVL_IO.aOutputSolValve.4 := valveSetting.4;
GVL_IO.aOutputSolValve.5 := valveSetting.5;
GVL_IO.aOutputSolValve.6 := valveSetting.6;
GVL_IO.aOutputSolValve.7 := valveSetting.7;

GVL_IO.aOutputSolValve.8 := valveSetting.8;
GVL_IO.aOutputSolValve.9 := valveSetting.9;
GVL_IO.aOutputSolValve.10 := valveSetting.10;
GVL_IO.aOutputSolValve.11 := valveSetting.11;
GVL_IO.aOutputSolValve.12 := valveSetting.12;
GVL_IO.aOutputSolValve.13 := valveSetting.13;
GVL_IO.aOutputSolValve.14 := valveSetting.14;
GVL_IO.aOutputSolValve.15 := valveSetting.15;

GVL_IO.aOutputSolValve.16 := valveSetting.16; 
GVL_IO.aOutputSolValve.17 := valveSetting.17;
GVL_IO.aOutputSolValve.18 := valveSetting.18;
GVL_IO.aOutputSolValve.19 := valveSetting.19;
//GVL_IO.aOutputSolValve.20 := valveSetting.20;

END_FUNCTION_BLOCK

// ---- POUs/P60_UpdatePV.TcPOU
PROGRAM P60_UpdatePV
VAR
	i: INT;
END_VAR

FOR i:=1 TO E_aAnalogInputIO_Index.E_PV_EPC_04 DO
	IF 0.0 < GVL_IO.aMaxValueController[i]  THEN		
		GVL_IO.aController_PV[i] := (GVL_IO.aAnalogInputIO[i] / GVL_CONSTANT.EL3064MaxValueH) * GVL_IO.aMaxValueController[i];
	END_IF
END_FOR

GVL_IO.aController_PV[E_aAnalogInputIO_Index.E_PV_Susceptor_Temp] := WORD_TO_REAL(GVL_IO.wE3508_PV);
GVL_IO.aController_PV[E_aAnalogInputIO_Index.E_PV_Reactor_Pressure] := WORD_TO_REAL(GVL_IO.wIqPlus_CDG2_PV);
GVL_IO.aController_PV[E_aAnalogInputIO_Index.E_PV_susceptorRotation] := GVL_IO.nRotation_Converted_PV;

END_PROGRAM

// ---- POUs/P70_Interface.TcPOU
PROGRAM P70_Interface
VAR
END_VAR

//

END_PROGRAM

// ---- POUs/P91_Monitoring.TcPOU
PROGRAM P91_Monitoring
VAR
	TimeCycle			: TON;
	i 					: INT;
	idx					: INT;
	
	(*Utility Input*)
	bUtilityFault		: BYTE;	
	JhValue_DOR: REAL;
	JhValue_EXHAUST: REAL;
END_VAR

//jhkang

(* Read from Utility Device*)

//jhkang butilityFault 는 어떤 것인가?
bUtilityFault.0		:= GVL_IO_GAS_CABINET.DI_05_ExternalH2GasCabinetFault;
bUtilityFault.1		:= GVL_IO_GAS_CABINET.DI_05_ExternalH2SGasCabinetFault;
bUtilityFault.2		:= GVL_IO_GAS_CABINET.DI_05_ExternalH2SeGasCabinetFault;
bUtilityFault.3		:= GVL_IO_GAS_CABINET.DI_05_ExternalUserInputAlarm;

TimeCycle(IN:=TRUE, PT:=T#100MS); // 100MS Refresh Reading Time
IF TimeCycle.Q THEN
	TimeCycle(IN:=FALSE);
	_DOR_EXHAUST();
	// Reactor Ultimate Pressure Gauge
	GVL_IO.aMonitoring_PV[1] := GVL_IO.aAnalogInputIO[E_aAnalogInputIO_Index.E_PV_Ultimate_Pressure] / GVL_CONSTANT.EL3064MaxValue * 10; //Ultimate Pressure 10Torr, 0~10V, Cal. x10
	GVL_IO.aMonitoring_PV[2] := JhValue_EXHAUST;
	GVL_IO.aMonitoring_PV[3] := JhValue_DOR;
	GVL_IO.aMonitoring_PV[4] := GVL_IO.aAnalogInputIO[E_aAnalogInputIO_Index.E_PV_GAS_Pressure_N2] / GVL_CONSTANT.EL3064MaxValue * 10; //N2 Cal. 6.89 bar  
	GVL_IO.aMonitoring_PV[5] := GVL_IO.aAnalogInputIO[E_aAnalogInputIO_Index.E_PV_GAS_Pressure_H2] / GVL_CONSTANT.EL3064MaxValue * 10; //H2 Cal. 6.89 bar
	GVL_IO.aMonitoring_PV[6] := GVL_IO.aAnalogInputIO[E_aAnalogInputIO_Index.E_PV_GAS_Pressure_H2S] / GVL_CONSTANT.EL3064MaxValue * 10; //NH3 Cal. 6.89 bar
	GVL_IO.aMonitoring_PV[7] := GVL_IO.aAnalogInputIO[E_aAnalogInputIO_Index.E_PV_GAS_Pressure_H2Se] / GVL_CONSTANT.EL3064MaxValue * 10; // Cal. 6.89 bar
	GVL_IO.aMonitoring_PV[8] := GVL_IO.aAnalogInputIO[E_aAnalogInputIO_Index.E_PV_CoolingWafer_SH] * 0.1; //  // PT100, Shower Head, Cal. 0.1
	GVL_IO.aMonitoring_PV[9] := GVL_IO.aAnalogInputIO2[1] / GVL_CONSTANT.EL3102MAxValue * 10;
	GVL_IO.aMonitoring_PV[10] := GVL_IO.aAnalogInputIO2[2] / GVL_CONSTANT.EL3102MAxValue * 10 ; 
	GVL_IO.aMonitoring_PV[11] := WORD_TO_REAL(P11_E3508.wE3508_PowerRate)*0.1; //divided to 10 PowerRate
	GVL_IO.aMonitoring_PV[12] := P12_IQ_PLUS.wByteValvePosition_PV_Monitoring;
	GVL_IO.aMonitoring_PV[13] := P14_ThermalBath.rTemperature_PV[1];
	GVL_IO.aMonitoring_PV[14] := P14_ThermalBath.rTemperature_PV[2];
	GVL_IO.aMonitoring_PV[15] := P14_ThermalBath.rTemperature_PV[3];
	GVL_IO.aMonitoring_PV[16] := P14_ThermalBath.rTemperature_PV[4];
	
	// A Line으로 들어가는 MFC 총량
	
	GVL_IO.aMonitoring_PV[17] := GVL_IO.aController_PV[E_aAnalogInputIO_Index.E_PV_MFC_01];
	
	IF  GVL_IO_VALVE.DO_00_V17GasH2SeManifoldRun = TRUE THEN
		GVL_IO.aMonitoring_PV[17]:=GVL_IO.aMonitoring_PV[17] + GVL_IO.aController_PV[E_aAnalogInputIO_Index.E_PV_MFC_03];
	END_IF
		IF  GVL_IO_VALVE.DO_00_V18GasH2SManifoldRun = TRUE THEN
		GVL_IO.aMonitoring_PV[17]:=GVL_IO.aMonitoring_PV[17] + GVL_IO.aController_PV[E_aAnalogInputIO_Index.E_PV_MFC_04];
	END_IF
		IF  GVL_IO_VALVE.DO_00_V19Source_4ChalcogenManifoldRun = TRUE THEN
		GVL_IO.aMonitoring_PV[17]:=GVL_IO.aMonitoring_PV[17] + GVL_IO.aController_PV[E_aAnalogInputIO_Index.E_PV_MFC_08];
	END_IF
	
	
	
	
	
	GVL_IO.aMonitoring_PV[18] := GVL_IO.aController_PV[E_aAnalogInputIO_Index.E_PV_MFC_02];
	IF  GVL_IO_VALVE.DO_00_V14Source_1TMInManifoldRun = TRUE THEN
		GVL_IO.aMonitoring_PV[18]:=GVL_IO.aMonitoring_PV[18] + GVL_IO.aController_PV[E_aAnalogInputIO_Index.E_PV_MFC_05];
	END_IF
	IF  GVL_IO_VALVE.DO_00_V15Source_2TMGaManifoldRun = TRUE THEN
		GVL_IO.aMonitoring_PV[18]:=GVL_IO.aMonitoring_PV[18] + GVL_IO.aController_PV[E_aAnalogInputIO_Index.E_PV_MFC_06];
	END_IF
	IF  GVL_IO_VALVE.DO_00_V16Source_3DMSeManifoldRun = TRUE THEN
		GVL_IO.aMonitoring_PV[18]:=GVL_IO.aMonitoring_PV[18] + GVL_IO.aController_PV[E_aAnalogInputIO_Index.E_PV_MFC_07];
	END_IF
END_IF

ACTION _DOR_EXHAUST:
GVL_SEQUENCE.FB_DOR_PRESSURE_AVG(newValue:=F_GetDorPressure(GVL_IO.aAnalogInputIO[E_aAnalogInputIO_Index.E_PV_DOR_PRESSURE]),Output=>JhValue_DOR);
GVL_SEQUENCE.FB_EXHAUST_AVG(newValue:=F_GetDorPressure(GVL_IO.aAnalogInputIO[E_aAnalogInputIO_Index.E_PV_Exhaust_Pressure]),Output=>JhValue_EXHAUST);
END_ACTION

END_PROGRAM

// ---- DEVICE/LINE HEATER/FB_LINE_HEATER_MANAGER.TcPOU
FUNCTION_BLOCK FB_LINE_HEATER_MANAGER
VAR_INPUT
	sendMessage			:ST_Modbus_Send_Frame;
END_VAR
VAR_OUTPUT
	bWriteError			:BOOL; 
	bReadError			:BOOL;
	bSendBufferusFull	:BOOL;
	bConnectError 		: BOOL;
	
	RData_Module_1	:ST_LineHeater_Data;
	RData_Module_2	:ST_LineHeater_Data;
END_VAR
VAR
	fbModbus_Master		:ModbusRtuMasterV2_KL6x22B;
	ReconnectTon		:TON;
	DataReadTon			:TON;
	bWriteExecute		:BOOL;
	bReadExecute		:BOOL;
	arrReceivedBuffer 	:ARRAY [0..24] OF WORD;
	arrSendBuffer 		:ARRAY [0..99] OF WORD;
	
	nModbusRead_Start_ADDR	:BYTE;
	nModbusWrite_Start_ADDR	:WORD;
	nReadExecuteCount		:UDINT;
		
	fbStructModbusSend:FB_MODBUS_SEND_FIFO;
	stOutput:ST_MODBUS_SEND_FRAME;
	
	nWriteQuantity		:WORD;
	fallEdge			:F_TRIG;
	backCount			: UDINT;
	nCycle				: UDINT;
	ReceivedTime		: UDINT;
	ResendTon			: Ton;
	rinedge				: R_TRIG;
	WriteCount			: INT;
	CheckLoad			: REAL;
	ErrorCount			: INT;
	BufferCount_Zefo	: INT;
	fTrigWriteComplete	: F_TRIG;
	ReReadTon: TON;
	ReReadTrig			: BOOL;
	
	ReadInputRegsBusy		: BOOL;
	ReadInputRegsError		: BOOL;
	WriteSingleRegisterBusy	: BOOL;
	WriteSingleRegisterError: BOOL;
	nModbusWrite_UniD: BYTE;
	ReadErrorID: Tc2_ModbusRTU.MODBUS_ERRORS;
	ReadLength: UINT;
	bReadSend: BOOL;
END_VAR

IF  ReadInputRegsError =FALSE THEN
	_Case();
	_CheckSendData();
ELSE
	ReconnectTon(IN:=ReconnectTon.Q=FALSE AND TRUE,pt:=T#1S);
	
	IF ReconnectTon.Q THEN
		
		ErrorCount := ErrorCount +1;
		
		IF ReadInputRegsError = TRUE THEN
			bReadExecute:=NOT bReadExecute;
		END_IF
		
	END_IF
END_IF

_ModbusFunction();

fbStructModbusSend();

bConnectError:= ReadInputRegsError;

ACTION _Case:
IF ReadInputRegsBusy = TRUE OR ReadInputRegsError = TRUE AND bWriteExecute = FALSE AND WriteSingleRegisterBusy = FALSE  THEN
	bReadExecute := FALSE;
	IF ReadInputRegsError = TRUE THEN
		bReadError:=TRUE;
	END_IF
END_IF

(*Copy Data*)
IF (ReadInputRegsBusy = FALSE AND ReadInputRegsError = FALSE)  THEN
	IF (fbModbus_Master.cbRead = 48 )  (*AND (arrReceivedBuffer[4] <> 0)*) THEN
		
//	IF arrReceivedBuffer[4] = 0 THEN
//		BufferCount_Zefo:=BufferCount_Zefo +1 ; 
//	END_IF

		CASE nReadExecuteCount OF
			1:MEMCPY(ADR(RData_Module_1),ADR(arrReceivedBuffer),SIZEOF(RData_Module_1));
				ReceivedTime :=nCycle;
				nCycle:=0;
			2:MEMCPY(ADR(RData_Module_2),ADR(arrReceivedBuffer),SIZEOF(RData_Module_2));
		END_CASE
	END_IF
	
END_IF
	nCycle:=nCycle+1;

(*Change Address*)
IF ReadInputRegsBusy = FALSE  AND ReadInputRegsError = FALSE  AND fbStructModbusSend.nBufferCount = 0 AND bWriteExecute = FALSE AND WriteSingleRegisterBusy = FALSE THEN
	DataReadTon(IN:=TRUE,pT:=T#500MS);
	IF DataReadTon.Q THEN
		
		nReadExecuteCount:=nReadExecuteCount+1;
		DataReadTon(IN:=FALSE);
		bReadExecute:=TRUE;
		
		MEMSET(ADR(arrReceivedBuffer),0,SIZEOF(arrReceivedBuffer));
		
		CASE nReadExecuteCount OF
			1:
				nModbusRead_Start_ADDR:=1;
			2:
				nModbusRead_Start_ADDR:=2;
				
			3:
				nReadExecuteCount:=0;
		ELSE
			nReadExecuteCount:=0;
			bReadExecute:=false;
		END_CASE
	END_IF
END_IF
END_ACTION

ACTION _CheckSendData:
IF WriteSingleRegisterBusy = FALSE OR WriteSingleRegisterError = TRUE THEN
	bWriteExecute := FALSE;
END_IF

IF fbStructModbusSend.nBufferCount > 0 AND bWriteExecute = FALSE AND WriteSingleRegisterBusy = FALSE THEN
	ResendTon(IN:=TRUE,pt:=T#150MS);
	rinedge(CLK:=ResendTon.Q);
	IF rinedge.q THEN
		ResendTon(IN:=FALSE);
		fbStructModbusSend.A_Remove(stOutput=>stOutput);
		
		nWriteQuantity:=stOutput.sendQuantity;
		nModbusWrite_UniD:=stOutput.UnitID;
		nModbusWrite_Start_ADDR:=stOutput.StartAddress;
		MEMCPY(ADR(arrSendBuffer),ADR(stoutput.SendData),SIZEOF(stoutput.SendData));
		
		bWriteExecute:=TRUE;
		nReadExecuteCount:=0;
		rinedge(CLK:=FALSE);
		ReReadTrig:=FALSE;
	END_IF
END_IF
END_ACTION

ACTION _ModbusFunction:
//Write the Regs to Modbus Server Function16
IF ReadInputRegsBusy = FALSE THEN
	fbModbus_Master.WriteSingleRegister(
		UnitID:= nModbusWrite_UniD, 
		Quantity:= nWriteQuantity, 
		MBAddr:= nModbusWrite_Start_ADDR, 
		cbLength:= SIZEOF(arrSendBuffer),
		pMemoryAddr:= ADR(arrSendBuffer),
		AuxQuantity:= , 
		AuxMBAddr:= , 
		AuxcbLength:= , 
		pAuxMemoryAddr:= , 
		Execute:= bWriteExecute,
		Timeout:= T#1S , 
		BUSY=>WriteSingleRegisterBusy ,
		Error=>WriteSingleRegisterError , 
		ErrorId=> , 
		cbRead=> );
END_IF

IF WriteSingleRegisterError THEN
	WriteCount:=WriteCount+1;
END_IF

IF WriteSingleRegisterBusy = FALSE  THEN
	//Read the Regs FROM Modbus Server Function3
	fbModbus_Master.ReadInputRegs(
		UnitID:= nModbusRead_Start_ADDR, // 온도 콘트롤러 ID 
		Quantity:= 24, // 통신 데이터 사이즈
		MBAddr:= 16#03E8, //레지스터 주소
		cbLength:= SIZEOF(arrReceivedBuffer) , 
		pMemoryAddr:= ADR(arrReceivedBuffer),
		Execute:= bReadExecute,
		Timeout:= T#1S , 
		BUSY=>ReadInputRegsBusy ,
		Error=> ReadInputRegsError,
		ErrorId=>ReadErrorID, 
		cbRead=>ReadLength );	
END_IF
END_ACTION

ACTION _SendModbusCommand:
IF fbStructModbusSend.nLoad < 90THEN
	IF 	fbStructModbusSend.nLoad > CheckLoad THEN 
		CheckLoad := fbStructModbusSend.nLoad;
	END_IF
	
	fbStructModbusSend.A_Add(stinput:=sendMessage);	
END_IF
END_ACTION

END_FUNCTION_BLOCK

// ---- DEVICE/LINE HEATER/FB_Modbus_Send_FIFO.TcPOU
FUNCTION_BLOCK FB_Modbus_Send_FIFO
VAR_INPUT
	stInput				:ST_Modbus_Send_Frame;
END_VAR
VAR_OUTPUT
	bExistMessage		:BOOL;
	nBufferCount		:UDINT;
	nLoad				:REAL;
	stOutput			:ST_Modbus_Send_Frame;
END_VAR
VAR
	ArrBuffer			:ARRAY[0..10000] OF BYTE;
	fbBuffer			:FB_MemRingBuffer;
	bOk					:BOOL;
	cbSize				:UDINT;
	
	nCurrentBuffer		:UDINT;
	BufferSize			:UINT;
END_VAR

bExistMessage := nBufferCount > 0;
BufferSize := SIZEOF(ArrBuffer);
nLoad :=  (UDINT_TO_REAL(fbBuffer.cbSize)/UDINT_TO_REAL(BufferSize)) * 100.0;;

ACTION A_Add:
fbBuffer.A_AddTail(	pWrite:=ADR(stInput),
					cbWrite:= SIZEOF( stInput ),
					pBuffer:= ADR( arrBuffer ),
					cbBuffer:= SIZEOF( arrBuffer ),
					bOk=> bOk,
					nCount => nBufferCount );
END_ACTION

ACTION A_Remove:
fbBuffer.A_RemoveHead(
						pRead:= ADR(stOutput ),
						cbRead:= SIZEOF( stOutput ),
						pBuffer:= ADR( arrBuffer ),
						cbBuffer:= SIZEOF( arrBuffer ),
						bOk=> bOk,
						nCount => nBufferCount );
END_ACTION

ACTION A_Reset:
MEMSET(ADR(ArrBuffer),0,SIZEOF(ArrBuffer));

fbBuffer.A_Reset(bOk=>bOk,
			nCount=>nBufferCount);			
			bExistMessage := nBufferCount > 0;
nLoad := fbBuffer.cbSize  / 200;
END_ACTION

END_FUNCTION_BLOCK

// ---- DEVICE/LINE HEATER/FUNCTION/F_Temp_Write_Set_Point.TcPOU
FUNCTION F_Temp_Write_Set_Point : ST_Modbus_Send_Frame
VAR_INPUT
	Module_Number:BYTE;
	CommandIndex:WORD;
	Write_Value:WORD;
END_VAR
VAR
END_VAR

F_Temp_Write_Set_Point := F_Temp_Write_Value(Module_Number:=Module_Number,
											Command_Index:=CommandIndex,
											Write_Value:=Write_Value);

END_FUNCTION

// ---- FUNCTION/F_State_All_Valve_Vent.TcPOU
FUNCTION F_State_All_Valve_Vent : bool
VAR_INPUT
END_VAR
VAR
END_VAR

F_State_All_Valve_Vent := GVL_IO_VALVE.DO_00_V01ChalcogenCarrierChange = FALSE  AND
				GVL_IO_VALVE.DO_00_V02MOCarreirChange = FALSE  AND
				GVL_IO_VALVE.DO_00_V03H2SeSourceChange = FALSE  AND
				GVL_IO_VALVE.DO_00_V04H2SSourceChange = FALSE  AND
				GVL_IO_VALVE.DO_00_V05Source_1TMInCarrierChange = FALSE  AND
				GVL_IO_VALVE.DO_00_V06Source_1TMInBypass = FALSE  AND
				GVL_IO_VALVE.DO_00_V07Source_2TMGaCarrierChange = FALSE  AND
				GVL_IO_VALVE.DO_00_V08Source_2TMGaBypass = FALSE  AND
				GVL_IO_VALVE.DO_00_V09Source_3DMSeCarrierChange = FALSE  AND
				GVL_IO_VALVE.DO_00_V10Source_3DMSeBypass = FALSE  AND
				GVL_IO_VALVE.DO_00_V11Source_4ChalcogenCarrierChange = FALSE  AND
				GVL_IO_VALVE.DO_00_V12Source_4ChalcogenBypass = FALSE AND
				GVL_IO_VALVE.DO_00_V13ReactorPurgeCarrierChange = FALSE AND
				GVL_IO_VALVE.DO_00_V14Source_1TMInManifoldRun = FALSE AND
				GVL_IO_VALVE.DO_00_V15Source_2TMGaManifoldRun = FALSE AND
				GVL_IO_VALVE.DO_00_V16Source_3DMSeManifoldRun = FALSE AND
				GVL_IO_VALVE.DO_00_V17GasH2SeManifoldRun = FALSE AND
				GVL_IO_VALVE.DO_00_V18GasH2SManifoldRun = FALSE ;

END_FUNCTION

// ---- FUNCTION/HEXSTR_TO_REAL_LHeaterPV.TcPOU
FUNCTION HEXSTR_TO_REAL_LHeaterPV : REAL
VAR_INPUT
	hStrTemperaturePV : STRING;
END_VAR
VAR
	hData			:UDINT;
	aData	: ARRAY[0..1]OF BYTE;
	bSwap	: BYTE;
	ptStrTemperature : POINTER TO INT;
	nTemperaturePV : INT;
END_VAR

//// Convert to Data Array from HexString
//hData := HEXSTR_TO_DATA(hStrTemperaturePV, ADR(aData), SIZEOF(aData));

////Swap Data
//bSwap := aData[0];
//aData[0] := aData[1];
//aData[1] := bSwap;

//ptStrTemperature := ADR(aData);
//nTemperaturePV := ptStrTemperature^;
//HEXSTR_TO_REAL_LHeaterPV := INT_TO_REAL(nTemperaturePV);

END_FUNCTION

// ---- POUs/FB_ControlRampGenerator.TcPOU
FUNCTION_BLOCK FB_ControlRampGenerator
VAR_INPUT
	input : RampGeneratorInput;
END_VAR
VAR
	state : E_RampGeneratorState := E_RampGeneratorState.End;
	rampGenerator : FB_CTRL_RAMP_GENERATOR;
	rampGeneratorParams	: ST_CTRL_RAMP_GENERATOR_PARAMS := (tTaskCycleTime := T#100MS, tCtrlCycleTime := T#100MS, fVeloPos := 0, fVeloNeg := 0);
END_VAR
VAR_OUTPUT
	rControlValue	: LREAL := 0;
	targetValueReached : BOOL := FALSE;
	isError : BOOL;
	eErrorID : E_CTRL_ERRORCODES;
END_VAR

IF input.restart = TRUE AND 0 <= input.rampTime AND rControlValue <> input.targetValue THEN
	state := E_RampGeneratorState.Init;
	input.restart := FALSE;
END_IF
	
CASE state OF
	E_RampGeneratorState.Init:
		IF 0 < input.rampTime THEN
			rampGeneratorParams.fVeloPos			:= ABS(input.targetValue - rControlValue) / input.rampTime * 0.1; (* in units per second *)
			rampGeneratorParams.fVeloNeg			:= rampGeneratorParams.fVeloPos; (* in units per second *)
			rampGenerator(bEnable := TRUE, fStart := rControlValue, fTarget:= input.targetValue, fOut => rControlValue, bValueReached => targetValueReached, bError => isError, eErrorID => eErrorID, stParams := rampGeneratorParams);
		ELSIF input.rampTime = 0 THEN
			rampGenerator(bEnable := FALSE, stParams := rampGeneratorParams);
			rampGeneratorParams.fVeloPos			:= input.targetValue; (* in units per second *)
			rampGeneratorParams.fVeloNeg			:= rampGeneratorParams.fVeloPos; (* in units per second *)
			rampGenerator(bEnable := TRUE, fStart := input.targetValue, fTarget:= input.targetValue, fOut => rControlValue, bValueReached => targetValueReached, bError => isError, eErrorID => eErrorID, stParams := rampGeneratorParams);
		END_IF
		state := E_RampGeneratorState.Run;
	
	E_RampGeneratorState.Run:
		rampGenerator(bEnable := TRUE, stParams := rampGeneratorParams, fOut => rControlValue, bValueReached => targetValueReached, bError => isError, eErrorID => eErrorID, stParams := rampGeneratorParams);
		IF targetValueReached = TRUE THEN
			state := E_RampGeneratorState.End;
		END_IF
		
	E_RampGeneratorState.End:
		rampGenerator(bEnable := FALSE, stParams := rampGeneratorParams, fOut => rControlValue);
END_CASE

END_FUNCTION_BLOCK
